    IF (_eRslt = E_PROGRESS.PROGRESS_DONE)
    THEN
      _XtsTransportCtrl.Cmd     := E_XTS_TRANSPORT_CTRL.CMD_TRANSPORT_START;
  
      IF (_XtsTransportState.State = E_XTS_TRANSPORT_STATE.TRANSPORT_START + E_PROGRESS.PROGRESS_ERROR)
      THEN
        _eState                             := E_PROGRESS.PROGRESS_ERROR;
        _TransportState                     := _XtsTransportState.State MOD E_PROGRESS.PROGRESS_ERROR;

        _stMsg.eType                        := E_MessageType.eMessageError;
        _stMsg.eSubdevice                   := e_Subdevice.Application_Work;
        _stMsg.iErrorNumber                 := _nErrorId;
        _stMsg.sText                        := concat(TO_STRING(_eState), ': ');
        _stMsg.sText                        := concat(_stMsg.sText, TO_STRING(_TransportState));
        f_MessageSet(_stMsg);
  
      ELSIF (_XtsTransportState.State = E_XTS_TRANSPORT_STATE.TRANSPORT_START + E_PROGRESS.PROGRESS_DONE)
      THEN
        _eState                             := E_PROGRESS.PROGRESS_PREPARE;
        _TransportState                     := _XtsTransportState.State MOD E_PROGRESS.PROGRESS_DONE;

        IF (_MessageLevel > E_MessageType.eMessageError)
        THEN
          _stMsg.eType                      := E_MessageType.eMessageInfo;
          _stMsg.eSubdevice                 := e_Subdevice.Application_Work;
          _stMsg.iErrorNumber               := 0;
          _stMsg.sText                      := concat(TO_STRING(_eState), ': ');
          _stMsg.sText                      := concat(_stMsg.sText, TO_STRING(_TransportState));
          f_MessageSet(_stMsg);
        END_IF
      END_IF
    END_IF

  E_PROGRESS.PROGRESS_PREPARE:
    _eRslt                                  := ListData(FALSE);
    IF (_eRslt = E_PROGRESS.PROGRESS_INIT)
    THEN
      _eState                               := E_PROGRESS.PROGRESS_STARTUP;
      _InfeedListCtrl.Cmd                   := e_list_ctrl.LIST_CTRL_NULL;

      _InfeedListDataInput.ProcessData.wTarget    := f_To_T_Process(TO_BYTE(_InstanceState[E_INSTANCE.INFEED].StationCount));
      _InfeedListDataInput.ProcessData.nProcessId := E_INSTANCE.SENDER_BUFFER_INFEED;
    END_IF     


  E_PROGRESS.PROGRESS_STARTUP:  // SENDER_BUFFER_INFEED sends the first batch of movers to BUFFER_INFEED
                                //  - after sending the first batch 
                                //    --> the transfersystem (ListData) may start writing entries into BUFFER_INFEED
    CASE _InstanceState[E_INSTANCE.SENDER_BUFFER_INFEED].State
    OF
    E_INSTANCE_STATE.DISABLED:

      CASE _InstanceState[E_INSTANCE.SENDER_BUFFER_INFEED].Progress
      OF
      E_PROGRESS.PROGRESS_BUSY:
        _eState                             := E_PROGRESS.PROGRESS_CHECK;
        _InfeedListCtrl.Cmd                 := e_list_ctrl.LIST_CTRL_ADD_TAIL;

        IF (_MessageLevel > E_MessageType.eMessageError)
        THEN
          _stMsg.eType                      := E_MessageType.eMessageInfo;
          _stMsg.eSubdevice                 := e_Subdevice.Application_Work;
          _stMsg.iErrorNumber               := 0;
          _stMsg.sText                      := concat(TO_STRING(_eState), ': ');
          _stMsg.sText                      := concat(_stMsg.sText, TO_STRING(e_Subdevice.Process_LinkedList_AddTail));
          f_MessageSet(_stMsg);
        END_IF
      END_CASE
    END_CASE
END_CASE
//-----------------------------------------------------------------------------
//-----------------------------------------------------------------------------
CASE _eState
OF
  E_PROGRESS.PROGRESS_CHECK:
    IF (_InfeedListState.State = e_list_state.LIST_STATE_ADD_TAIL + e_progress.PROGRESS_DONE)
    THEN
      _eState                                         := E_PROGRESS.PROGRESS_OCCUPIED;
      _InfeedListCtrl.Cmd                             := e_list_ctrl.LIST_CTRL_NULL;
      _InstanceCtrl[E_INSTANCE.PROCESS_CONDUCTOR].Cmd := E_INSTANCE_CMD.ENABLE;
      _InstanceCtrl[E_INSTANCE.BUFFER_INFEED].Cmd     := E_INSTANCE_CMD.ENABLE;


    ELSIF (_InfeedListState.State = e_list_state.LIST_STATE_ADD_TAIL + e_progress.PROGRESS_ERROR)
    THEN
      _eState                               := E_PROGRESS.PROGRESS_ERROR;
    END_IF 
END_CASE
//-----------------------------------------------------------------------------
//-----------------------------------------------------------------------------
CASE _eState
OF
  E_PROGRESS.PROGRESS_OCCUPIED:
    IF NOT _bSwitchManual
    THEN
      _eState                               := E_PROGRESS.PROGRESS_WORKING;
    END_IF

    IF (_MessageLevel > E_MessageType.eMessageError)
    THEN
      _stMsg.eType                          := E_MessageType.eMessageInfo;
      _stMsg.eSubdevice                     := e_Subdevice.Application_Work;
      _stMsg.iErrorNumber                   := 0;
      _stMsg.sText                          := concat(TO_STRING(_eState), ': ');
      f_MessageSet(_stMsg);
    END_IF
END_CASE
//-----------------------------------------------------------------------------
//-----------------------------------------------------------------------------
CASE _eState
OF
  E_PROGRESS.PROGRESS_WORKING:
    FOR _eInst := E_INSTANCE.PROCESS_CONDUCTOR TO E_INSTANCE.SENDER_BUFFER_INFEED
    DO
      // handshakes to instances: 
      // - deconstruct this for your own implementation
      CASE _InstanceState[_eInst].State
      OF
        E_INSTANCE_STATE.DISABLED:
          CASE _InstanceState[_eInst].Progress
          OF
            E_PROGRESS.PROGRESS_BUSY:
            CASE _eInst
            OF
              e_instance.PROCESS_CONDUCTOR:

                CASE _InstanceState[e_instance.BUFFER_INFEED].State
                OF
                  E_INSTANCE_STATE.DETECTION:
                    _eRslt                  := ListData(FALSE);

                    IF NOT _bTicketCountOverride
                    THEN
                      IF (_nTicketCount < _nTicketCountEnd+1)
                      THEN
                        _InstanceCtrl[e_instance.PROCESS_CONDUCTOR].Cmd := E_INSTANCE_CMD.ENABLE;
                      END_IF
                    ELSE
                      _InstanceCtrl[e_instance.PROCESS_CONDUCTOR].Cmd   := E_INSTANCE_CMD.ENABLE;
                    END_IF
                END_CASE
            ELSE
                _InstanceCtrl[_eInst].Cmd   := E_INSTANCE_CMD.ENABLE;
            END_CASE
          END_CASE
      
        E_INSTANCE_STATE.ENABLED:
          CASE _InstanceState[_eInst].Progress
          OF
            E_PROGRESS.PROGRESS_OCCUPIED:
              _InstanceCtrl[_eInst].Cmd     := E_INSTANCE_CMD.PROCEED;
          END_CASE

        E_INSTANCE_STATE.WORKING:
          CASE _InstanceState[_eInst].Progress
          OF
            E_PROGRESS.PROGRESS_BUSY:
              _tonProcess [_eInst]
                              (IN           := FALSE, 
                               PT           := _tProcess[_eInst]);


              IF (_eInst > E_INSTANCE.OUTFEED_ROBOT_R2) OR
                 (_eInst < E_INSTANCE.OUTFEED_ROBOT_R1) OR
                 (_bSingleOutput) OR
                 NOT (_Ctrl.Variant = E_APP_VARIANT.VARIANT_OUTPUT_24)
              THEN
                _InstanceCtrl[_eInst].Cmd   := E_INSTANCE_CMD.WORK;
              ELSE
                IF (_InstanceState[E_INSTANCE.OUTFEED_ROBOT_R1].State = 
                    _InstanceState[E_INSTANCE.OUTFEED_ROBOT_R2].State )
                THEN
                  // in this example the outfeed instances are working in sync
                  _InstanceCtrl[_eInst].Cmd := E_INSTANCE_CMD.WORK;

                  IF (_MessageLevel > E_MessageType.eMessageError)
                  THEN
                    _stMsg.eSubdevice       := e_Subdevice.Application_Work;
                    _stMsg.iErrorNumber     := _eInst;
                    _stMsg.sText            := concat('E_INSTANCE.', TO_STRING(_eInst));
                    _stMsg.sText            := concat(_stMsg.sText , ': E_INSTANCE_CMD.');
                    _stMsg.sText            := concat(_stMsg.sText , TO_STRING(_InstanceCtrl[_eInst].Cmd));

                    f_MessageSet(_stMsg);
                  END_IF
                END_IF
              END_IF
      
      
            E_PROGRESS.PROGRESS_CHECK:
              _tonProcess [_eInst]
                              (IN           := TRUE, 
                               PT           := _tProcess[_eInst]);
      
              IF _tonProcess [_eInst].Q
              THEN
                _InstanceCtrl[_eInst].Cmd   := E_INSTANCE_CMD.FINISH;

                IF (_MessageLevel > E_MessageType.eMessageError)
                THEN
                  _stMsg.eSubdevice         := e_Subdevice.Application_Work;
                  _stMsg.iErrorNumber       := _eInst;
                  _stMsg.sText              := concat('E_INSTANCE.', TO_STRING(_eInst));
                  _stMsg.sText              := concat(_stMsg.sText , ': E_INSTANCE_CMD.');
                  _stMsg.sText              := concat(_stMsg.sText , TO_STRING(_InstanceCtrl[_eInst].Cmd));
                  f_MessageSet(_stMsg);
                END_IF
              END_IF
          END_CASE


        E_INSTANCE_STATE.FINISH:
          CASE _InstanceState[_eInst].Progress
          OF
            E_PROGRESS.PROGRESS_BUSY:
              _tonProcess [_eInst]
                              (IN           := FALSE, 
                               PT           := _tProcess[_eInst]);

              _InstanceCtrl[_eInst].Cmd     := E_INSTANCE_CMD.FINISH;

            E_PROGRESS.PROGRESS_OCCUPIED:
              _InstanceCtrl[_eInst].Cmd     := E_INSTANCE_CMD.PROCEED;

            E_PROGRESS.PROGRESS_DONE:
                _eRslt                      := ListData(_bRunListData);
                IF (_eRslt = E_PROGRESS.PROGRESS_DONE)
                THEN
                  _InstanceCtrl[_eInst].Cmd := E_INSTANCE_CMD.FINISH;
                END_IF
          END_CASE
        END_CASE
    END_FOR
END_CASE
//-----------------------------------------------------------------------------
//-----------------------------------------------------------------------------
Work                                        := _eState;
END_METHOD

PROPERTY WriteTimeVariant : bool
GET
WriteTimeVariant := _bWriteTimeVariant;
END_GET
SET
_bWriteTimeVariant := WriteTimeVariant;
END_SET
END_PROPERTY

PROPERTY XtsTransportCtrl : REFERENCE TO ST_XTS_TRANSPORT_CTRL
SET
_XtsTransportCtrl REF= XtsTransportCtrl;
END_SET
END_PROPERTY

PROPERTY XtsTransportState : REFERENCE TO ST_XTS_TRANSPORT_STATE
SET
_XtsTransportState REF= XtsTransportState;
END_SET
END_PROPERTY

END_FUNCTION_BLOCK

(* stored: Version 1.1.0.1
   POU fb_Application: Id {d837f1a6-2825-42ae-9093-3e866ef4fbe7}, SpecialFunc None
   Folder methods: Id {98770898-61ad-40e0-8965-baa3ce19544a}
   Folder properties: Id {176b5ab6-95e4-4dca-b119-abdd9161e273}
   Method Check: Id {da6dfb36-1549-4909-ac88-0380a0759b2d}
   Method Clear: Id {2792b871-ea89-4b49-8178-26d234aeeb5f}
   Method Cmd: Id {25875579-afe9-4bc4-939f-25fe2bdae97b}
   Property Ctrl: Id {7b5da87a-23ec-43c8-a367-1d3eb2b8f2b5}
   Set Set: Id {b73a2f8e-7976-4c7b-aecf-4cd90d0d4ad4}
   Method Disable: Id {6a1967ac-bfda-4bfa-aaf3-54c7dba01ffd}
   Method Enable: Id {51767aef-3d3b-4973-9946-b6ec66b91d19}
   Method Finish: Id {f38628f8-bdae-4a59-b8b6-47346bf9974d}
   Property Info: Id {d32a928f-d6e9-4f23-9e4b-2152b71bed6c}
   Set Set: Id {57dec8bb-0f39-4566-9050-9b6a93c0d5be}
   Method Init: Id {ab722eef-0388-45b6-85d1-7a5a0fed75bd}
   Property InstanceCtrl: Id {685a5388-b581-438e-b059-318e6201ef4a}
   Set Set: Id {e5362d7d-8cbe-44c5-a53a-2dee1c05e695}
   Property InstanceState: Id {378b4970-b9c5-445e-818c-d12a2f5feb53}
   Set Set: Id {f2193521-74d4-42fb-8546-0af204d63725}
   Property ListControl: Id {1c4143b8-9b74-4bbe-9901-707f144b47ed}
   Set Set: Id {2ff9a875-7b0c-4791-a66a-ea6c6613c46d}
   Method ListData: Id {931d9c3b-db15-4ce4-a9db-7473a9252434}
   Property ListInputData: Id {75bcf882-30e6-4f13-b766-cbf7836a4278}
   Set Set: Id {3c330000-dd49-45c2-be1f-5a224752c62c}
   Property ListState: Id {cdbd355f-e84b-4409-84d6-ceee3f21eefa}
   Set Set: Id {b96a6bd6-ff69-4c8b-b3f7-bfb1d713f3c7}
   Property MessageLevel: Id {75b3b401-3d18-42e5-90df-8cac469d9946}
   Get Get: Id {14e09632-b9f9-4924-bbbd-ec9781609fab}
   Set Set: Id {940048a6-54e6-4562-9da8-ed83616a9106}
   Method Proceed: Id {15b4c3e6-5b70-4afc-b74d-0d947ff3addc}
   Property State: Id {fdba28c5-fd22-4379-8205-51455c4503c8}
   Set Set: Id {6fb63032-c021-47b2-9672-c9607ad424c1}
   Method Work: Id {7d710bc9-4a53-44f9-8fb0-654ccbd1ea75}
   Property WriteTimeVariant: Id {e8b254ad-2acd-4568-be47-536881d1af43}
   Get Get: Id {2816ca48-f02c-47fb-b95e-2093e30cc385}
   Set Set: Id {a2a1c020-9c61-44a3-9e11-340ef8ff21b4}
   Property XtsTransportCtrl: Id {5f6cc21b-cb5f-47bb-b3e6-a1a78d9341a1}
   Set Set: Id {249b8b7a-2d2b-48ca-896c-4c360c3c6d7f}
   Property XtsTransportState: Id {3997ef1a-6333-4545-add0-c3aa6af11a49}
   Set Set: Id {c34f1112-ea2f-4e7e-b2a5-e988837777d5} *)
